// TwinCAT 3 PLC project PLC
// ProgramVersion: 3.1.4024.0
// libraries:
//   Tc2_Standard, * (Beckhoff Automation GmbH)
//   Tc2_System, * (Beckhoff Automation GmbH)
//   Tc3_Module, * (Beckhoff Automation GmbH)
// project tree:
//   GVLs/ GVL.TcGVL
//   / PlcTask.TcTTO
//   POUs/ MAIN.TcPOU
// real-time tasks:
//   TASK PlcTask: cycle T#10ms, priority 20, ADS port 350
// I/O:
//   DEVICE Device 1 (EtherCAT), AmsNetId 192.168.71.1.2.1
//     Term 1 (EK1100) [EK1100 EtherCAT Coupler (2A E-Bus)]
//       Term 2 (EL2809) [EL2809 16Ch. Dig. Output 24V, 0.5A]
//       Term 3 (EL9505) [EL9505 Power supply terminal 5V]
//       Term 4 (EL3751) [EL3751 1Ch. Ana. Input +/-30V, +/-20mA, RTD, Resistor Bridge, 24 bit, high precision]
//       Term 5 (EL9011) [EL9011 End Terminal]
// variable links:
//   PLC/PLC Instance <-> Device 1 (EtherCAT)/Term 1 (EK1100)/Term 2 (EL2809)
//     PlcTask Outputs/GVL.q_Led <-> Channel 1/Output
//   PLC/PLC Instance <-> Device 1 (EtherCAT)/Term 1 (EK1100)/Term 4 (EL3751)
//     PlcTask Inputs/GVL.i_Analog <-> PAI Samples 1/Samples[0]

CONFIGURATION PLC
    RESOURCE PLC ON TwinCAT3
        TASK PlcTask(INTERVAL := T#10ms, PRIORITY := 20);
        PROGRAM MAIN WITH PlcTask : MAIN;
    END_RESOURCE
END_CONFIGURATION

// ---- GVLs/GVL.TcGVL
VAR_GLOBAL
	i_Analog 	AT %I* :DINT;
	q_Led 		AT %Q* :BOOL;
END_VAR

// ---- POUs/MAIN.TcPOU
PROGRAM MAIN
VAR
	//Buffer
	Size 		:INT:=1000;
    Buffer_y 	:ARRAY[1..1000] OF REAL; 
    i 			:INT := 1; 
	
	//Heart bit
	HBIT		:INT:= 1;
END_VAR

//Fill buffer to python 
FOR i := (Size-1) TO 1 BY -1 DO
    Buffer_y[i+1] := Buffer_y[i]; 
END_FOR
Buffer_y[1] := DINT_TO_REAL(i_Analog); 

//Heart Bit
HBIT := HBIT + 1;
IF HBIT >= 100 THEN
	q_Led := NOT q_Led;
	HBIT := 0;
END_IF

END_PROGRAM
